(* PLC project  *)

PROGRAM BlocksXml
  VAR
    A : INT;
    B : INT;
    C : INT;
    D : INT;
  END_VAR

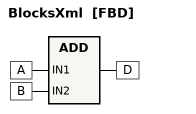
(* FBD diagram, written out as Structured Text *)
D := A + B;
END_PROGRAM
